// TIA Portal V20 export
DATA_BLOCK "BK01"   // DB87
// stored: MemoryReserve 100
   VAR
      "X10-1.BTM DIRECTION CHECK SENSOR" : Bool := TRUE;
      "X11-1.SEPA UNWINDER IONIZER TOP 2 POWER" : Bool := FALSE;
      "X12-1.SPARE" : Bool := FALSE;
      "X13-1.COMPENSATOR #1 LIMIT SENSOR(-)" : Bool := TRUE;
      "X14-1.COMPENSATOR #1 LIMIT SENSOR(+)" : Bool := TRUE;
      "X15-1.SPARE" : Bool := FALSE;
      "X16-1.SPARE" : Bool := FALSE;
      "X17-1.SAFETY PIN IDLE POSITION" : Bool := TRUE;
      "X10-2.TOP DIRECTION CHECK SENSOR" : Bool := FALSE;
      "X11-2.SEPA UNWINDER IONIZER BTM 2 POWER" : Bool := FALSE;
      "X12-2.SPARE" : Bool := FALSE;
      "X13-2.COMPENSATOR #1 HOME SENSOR" : Bool := TRUE;
      "X14-2.SPARE" : Bool := FALSE;
      "X15-2.SPARE" : Bool := FALSE;
      "X16-2.SPARE" : Bool := FALSE;
      "X17-2.SPARE" : Bool := FALSE;
   END_VAR
BEGIN
END_DATA_BLOCK
